(* IEC 61131-3 sources: structured-text/demo, 1 file *)

(* ---- thresh.st ---- *)
// LTL: [] ({not is_breaker_open and (meter_va > thresh)} -> () {is_breaker_open})
// LTL: [] {meter_va > 0}
FUNCTION THRESHOLD : BOOL
      VAR_INPUT
            meter_va : INT;
            is_breaker_open : BOOL;
            thresh : INT;
      END_VAR

      IF not is_breaker_open and (meter_va > thresh) THEN
            THRESHOLD := TRUE;
      ELSE
            THRESHOLD := FALSE;
      END_IF;
END_FUNCTION
